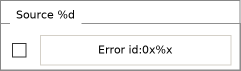
VISUALIZATION Event  // 241x71
VAR_IN_OUT
	Event:FB_SimpleAdsLogEvent;
END_VAR
    GroupBox (0,15 241x56)
        Button (120,20 111x30), "quit"
            tap Event.bQuit
        Textfield (40,20 71x30), "Event %d", text variable: Event.EventID
        Checkbox (10,20 31x30), variable: Event.bSetEvent
        Textfield (40,20 191x30), "Error id:0x%x", text variable: Event.ErrId, colour toggle: Event.Error, invisible if: NOT Event.Error
    Textfield (10,0 71x30), "Source %d", text variable: Event.SourceID
END_VISUALIZATION

(* stored: Version 1.1.0.1, ProductVersion 3.1.4024.11
   Visu Event: Id {9e8fd7c5-0447-0282-3192-b4ff9d6e4469} *)
